(* Logix 5000 project; controller SpineControl2 vendor 1 type 14 code 155 rev 20.12; software revision 20.01 *)

TASK MainTask (continuous, watchdog 500 ms) : MainProgram

MODULES
   Local : vendor 1 type 14 code 155 (PointIO 0, rev 20.12)
      Motor_Driver : vendor 1 type 37 code 28 (Ethernet 192.168.1.5, rev 1.1, MotionDiagnostics RPI 1 ms, MotionSync RPI 1 ms)
      Discrete_IO : Embedded (PointIO 1, rev 20.11, Output RPI 20 ms)
END_MODULES

VAR_GLOBAL   (* controller tags *)
   m_Accel_Jerk : DINT := 1;
   m_Accel_Rate : DINT := 2;
   m_Calc_Data : DINT;
   m_Decel_Jerk : DINT := 1;
   m_Decel_Rate : DINT := 2;
   m_Event_Dist : DINT;
   m_Lock_Position : DINT;
   m_MAH : MOTION_INSTRUCTION;
   m_MAM : MOTION_INSTRUCTION;
   m_MSF : MOTION_INSTRUCTION;
   m_MSO : MOTION_INSTRUCTION;
   m_Position : DINT := 50;
   m_Speed : DINT := 5;
   m_Type : DINT;
   motor1 : AXIS_CIP_DRIVE;
   motor_Enable : BOOL := 1;
   Motor_Group : MOTION_GROUP;
   move2Home : BOOL;
   sock_Accept_Connection : MESSAGE;
   sock_Create : MESSAGE;
   start_Motion : BOOL;
   start_Socket : BOOL;
END_VAR

PROGRAM MainProgram   (* main routine MainRoutine *)

ROUTINE MainRoutine   (* ladder *)
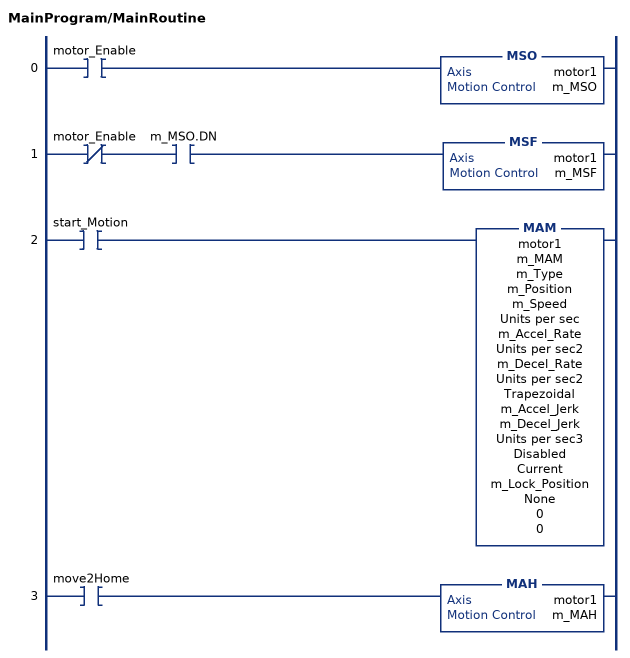
   0: XIC(motor_Enable)MSO(motor1,m_MSO);
   1: XIO(motor_Enable)XIC(m_MSO.DN)MSF(motor1,m_MSF);
   2: XIC(start_Motion)MAM(motor1,m_MAM,m_Type,m_Position,m_Speed,Units per sec,m_Accel_Rate,Units per sec2,m_Decel_Rate,Units per sec2,Trapezoidal,m_Accel_Jerk,m_Decel_Jerk,Units per sec3,Disabled,Current,m_Lock_Position,None,0,0);
   3: XIC(move2Home)MAH(motor1,m_MAH);
END_ROUTINE

ROUTINE socket_Initialize   (* ladder *)
// Initializes the socket connection.
// Windows program must connect before timeout time.
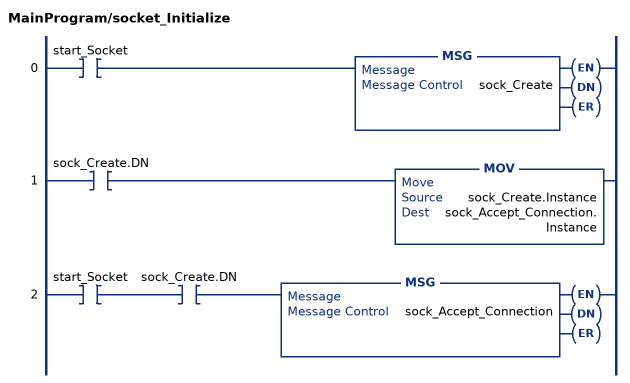
   0: XIC(start_Socket)MSG(sock_Create);
   1: XIC(sock_Create.DN)MOV(sock_Create.Instance,sock_Accept_Connection.Instance);
   2: XIC(start_Socket)XIC(sock_Create.DN)MSG(sock_Accept_Connection);
END_ROUTINE
END_PROGRAM
